// TwinCAT 3 PLC project PRG_HMIElements
// Title: B_HMIElements
// Company: RafalOS
// Author: Rafał Osajda
// ProjectVersion: 0.0.0.4
// ProgramVersion: 3.1.4024.0
// libraries:
//   B_Base, * (RafalOS)
//   B_Base_HMI_Connector, * (RafalOS)
//   Tc2_Standard, * (Beckhoff Automation GmbH)
//   Tc2_System, * (Beckhoff Automation GmbH)
//   Tc3_Module, * (Beckhoff Automation GmbH)
// project tree:
//   GVLs/ GVL_HMIEConstans.TcGVL (not stored)
//   / PlcTask.TcTTO
//   POUs Compilation/ PRG_Compilation.TcPOU
//   POUs/01A_Button/ FB_HMIEButton.TcPOU, ITF_HMIEButton.TcIO (not stored), ITF_HMIEButton_HMI_Connector.TcIO, ITF_HMIEButton_HMI_Init.TcIO (not stored)
//   POUs/01B_ButtonHMI/ FB_HMIEButton_HMI.TcPOU, ITF_HMIEButton_HMI.TcIO
//   POUs/02A_Menu/ FB_HMIEMenu.TcPOU, ITF_HMIEMenu_HMI_Connector.TcIO, ITF_HMIEMenu_HMI_Init.TcIO, ITF_HMIEMenu.TcIO
//   POUs/02B_MenuHMI/ FB_HMIEMenu_HMI.TcPOU, ITF_HMIEMenu_HMI.TcIO

CONFIGURATION PRG_HMIElements
    RESOURCE PLC ON TwinCAT3
        TASK PlcTask(INTERVAL := T#10ms, PRIORITY := 20);
        PROGRAM PRG_Compilation WITH PlcTask : PRG_Compilation;
    END_RESOURCE
END_CONFIGURATION

// ---- POUs/01A_Button/ITF_HMIEButton_HMI_Connector.TcIO
(*			
	RafalOS
	Rafał Osajda		12.11.2025		TC 4024.66
	Zbiór metod umożliwiające odczyt danych z hmi 
*)
INTERFACE ITF_HMIEButton_HMI_Connector EXTENDS ITF_BaseComponent_HMI_Connector

END_INTERFACE

// ---- POUs/01B_ButtonHMI/ITF_HMIEButton_HMI.TcIO
(*			
	RafalOS
	Rafał Osajda		12.11.2025		TC 4024.66
	interfejs potrzebny w HMI
*)
INTERFACE ITF_HMIEButton_HMI EXTENDS ITF_BaseComponent_HMI

END_INTERFACE

// ---- POUs/02A_Menu/ITF_HMIEMenu_HMI_Connector.TcIO
(*			
	RafalOS
	Rafał Osajda		12.11.2025		TC 4024.66
	Zbiór metod umożliwiające odczyt danych z hmi 
*)
INTERFACE ITF_HMIEMenu_HMI_Connector EXTENDS ITF_BaseControlElement_HMI_Connector

END_INTERFACE

// ---- POUs/02A_Menu/ITF_HMIEMenu_HMI_Init.TcIO
(*			
	RafalOS
	Rafał Osajda		12.11.2025		TC 4024.66
	interfejs do przekazywania przy tworzeniu elementów
*)
INTERFACE ITF_HMIEMenu_HMI_Init EXTENDS ITF_BaseControlElement, ITF_HMIEMenu_HMI_Connector

END_INTERFACE

// ---- POUs/02A_Menu/ITF_HMIEMenu.TcIO
INTERFACE ITF_HMIEMenu EXTENDS ITF_BaseControlElement

METHOD PUBLIC GetNumberOfActriveScreen : INT
VAR_INPUT
END_VAR
END_METHOD

METHOD IsActiveButton : BOOL
VAR_INPUT
	iButton		: INT;	//numer przycisku
	bIN			: BOOL;
END_VAR
END_METHOD

METHOD PUBLIC IsChangePage : BOOL
VAR_INPUT
END_VAR
END_METHOD

METHOD IsEnableButton : BOOL
VAR_INPUT
	iButton		: INT;	//numer przycisku
	bIN			: BOOL;
END_VAR
END_METHOD

METHOD IsVisibleButton : BOOL
VAR_INPUT
	iButton		: INT;	//numer przycisku
	bIN			: BOOL;
END_VAR
END_METHOD

METHOD PUBLIC ResetChangePage
VAR_INPUT
END_VAR
END_METHOD

METHOD SetActiveButton : BOOL
VAR_INPUT
	iButton		: INT;	//numer przycisku
	bIN			: BOOL;
END_VAR
END_METHOD

METHOD SetEnableButton : BOOL
VAR_INPUT
	iButton		: INT;	//numer przycisku
	bIN			: BOOL;
END_VAR
END_METHOD

METHOD SetVisibleButton : BOOL
VAR_INPUT
	iButton		: INT;	//numer przycisku
	bIN			: BOOL;
END_VAR
END_METHOD

(*			
	RafalOS
	Rafał Osajda		11.11.2025		TC 4024.66
	testuje czy jest coś naciśnięte w menu i przełącza
*)
METHOD PUBLIC Testing : BOOL
END_METHOD

END_INTERFACE

// ---- POUs/02B_MenuHMI/ITF_HMIEMenu_HMI.TcIO
(*			
	RafalOS
	Rafał Osajda		12.11.2025		TC 4024.66
	interfejs potrzebny w HMI
*)
INTERFACE ITF_HMIEMenu_HMI EXTENDS ITF_BaseComponent_HMI

END_INTERFACE

// ---- POUs Compilation/PRG_Compilation.TcPOU
PROGRAM PRG_Compilation
VAR
	fbButton		: FB_HMIEButton;
	fbButtonHMI		: FB_HMIEButton_HMI (itfButton := fbButton);
	fbMenu			: FB_HMIEMenu;
	fbMenuHMI		: FB_HMIEMenu_HMI (itfMenu := fbMenu);
END_VAR

END_PROGRAM

// ---- POUs/01A_Button/FB_HMIEButton.TcPOU
FUNCTION_BLOCK FB_HMIEButton EXTENDS FB_BaseComponent IMPLEMENTS ITF_HMIEButton, ITF_HMIEButton_HMI_Init
VAR
	bContact			: BOOL;
	bActive				: BOOL;	//wybrany
	bVisible			: BOOL; //widoczny
	bEnable				: BOOL; //wlaczony
END_VAR

METHOD PUBLIC IsActive : BOOL
VAR_INPUT
END_VAR
IsActive		:= THIS^.bActive;
END_METHOD

METHOD PUBLIC IsEnable : BOOL
VAR_INPUT
END_VAR
IsEnable		:= THIS^.bEnable;
END_METHOD

METHOD PUBLIC IsPressed : BOOL
VAR_INPUT
END_VAR
IsPressed		:= THIS^.bContact;
END_METHOD

METHOD PUBLIC IsVisible : BOOL
VAR_INPUT
END_VAR
IsVisible		:= THIS^.bVisible;
END_METHOD

METHOD PUBLIC SetActive
VAR_INPUT
	bIN: BOOL;
END_VAR
THIS^.bActive		:= bIN;
END_METHOD

METHOD PUBLIC SetEnable
VAR_INPUT
	bIN: BOOL;
END_VAR
THIS^.bEnable		:= bIN;
END_METHOD

METHOD PUBLIC SetPressed
VAR_INPUT
	bIN: BOOL;
END_VAR
THIS^.bContact		:= bIN;
END_METHOD

METHOD PUBLIC SetVisible
VAR_INPUT
	bIN: BOOL;
END_VAR
THIS^.bVisible		:= bIN;
END_METHOD

END_FUNCTION_BLOCK

// ---- POUs/01B_ButtonHMI/FB_HMIEButton_HMI.TcPOU
FUNCTION_BLOCK FB_HMIEButton_HMI EXTENDS FB_BaseComponent_HMI IMPLEMENTS ITF_HMIEButton_HMI
VAR
	itfButton			: ITF_HMIEButton_HMI_Connector;
END_VAR

METHOD FB_init : BOOL
VAR_INPUT
	bInitRetains : BOOL; // if TRUE, the retain variables are initialized (warm start / cold start)
	bInCopyCode : BOOL;  // if TRUE, the instance afterwards gets moved into the copy code (online change)
	itfButton			: ITF_HMIEButton_HMI_Init;
END_VAR
THIS^.itfButton := itfButton;
//Przypisanie do elementów z biblioteki
THIS^.itfBaseLoggerElementConnector		:= itfbutton;
THIS^.itfBaseComponentConnector			:= itfbutton;

//
THIS^.itfBaseLoggerConnector			:= itfBaseLoggerConnector;

IF (THIS^.itfButton <> 0 AND
	THIS^.itfBaseLoggerElementConnector <> 0 AND
	THIS^.itfBaseComponentConnector	<> 0 AND
	THIS^.itfBaseLoggerConnector <> 0) THEN
	THIS^.bIsInit						:= TRUE;
END_IF
END_METHOD

END_FUNCTION_BLOCK

// ---- POUs/02A_Menu/FB_HMIEMenu.TcPOU
FUNCTION_BLOCK FB_HMIEMenu EXTENDS FB_BaseControlElement IMPLEMENTS ITF_HMIEMenu, ITF_HMIEMenu_HMI_Init
VAR
	arrButtons				: ARRAY [0..GVL_HMIEConstans.MAX_NUMBER_OF_BUTTON_IN_MENU] OF ITF_HMIEButton;
	iNumberOfButton			: INT := -1;	//ilosć przycisków w menu
	iActiveButton			: INT;	//numer aktywnego przycisku
	iActiveButtonPrev		: INT;
	bChangePage				: BOOL; //zmiana strony
END_VAR

METHOD PUBLIC AddButton : BOOL
VAR_INPUT
	fbButton			: ITF_HMIEButton;
END_VAR
IF (THIS^.iNumberOfButton + 1 <= GVL_HMIEConstans.MAX_NUMBER_OF_BUTTON_IN_MENU) THEN
	THIS^.iNumberOfButton := THIS^.iNumberOfButton + 1;
	THIS^.arrButtons [THIS^.iNumberOfButton] := fbButton;
	THIS^.arrButtons [THIS^.iNumberOfButton].SetEnable (bIN := TRUE);
	THIS^.arrButtons [THIS^.iNumberOfButton].SetVisible (bIN := TRUE);
	THIS^.AddComponent (itfComponent := fbButton);
	AddButton := TRUE;
ELSE
	AddButton := FALSE;
END_IF
END_METHOD

METHOD PUBLIC GetNumberOfActrivePreviewScreen : INT
VAR_INPUT
END_VAR
GetNumberOfActrivePreviewScreen := THIS^.iActiveButtonPrev;
END_METHOD

METHOD PUBLIC GetNumberOfActriveScreen : INT
VAR_INPUT
END_VAR
GetNumberOfActriveScreen := THIS^.iActiveButton;
END_METHOD

METHOD PUBLIC GetTitleOfActivePage : WSTRING
VAR_INPUT
END_VAR
//GetTitleOfActivePage := this^.arrButtons [this^.iActiveButton].GetName ();
END_METHOD

METHOD IsActiveButton : BOOL
VAR_INPUT
	iButton		: INT;	//numer przycisku
	bIN			: BOOL;
END_VAR
IsActiveButton	:= THIS^.arrButtons [iButton].IsActive ();
END_METHOD

METHOD PUBLIC IsChangePage : BOOL
VAR_INPUT
END_VAR
IsChangePage := THIS^.bChangePage;
END_METHOD

METHOD IsEnableButton : BOOL
VAR_INPUT
	iButton		: INT;	//numer przycisku
	bIN			: BOOL;
END_VAR
IsEnableButton	:= THIS^.arrButtons [iButton].IsEnable ();
END_METHOD

METHOD IsVisibleButton : BOOL
VAR_INPUT
	iButton		: INT;	//numer przycisku
	bIN			: BOOL;
END_VAR
IsVisibleButton	:= THIS^.arrButtons [iButton].IsVisible ();
END_METHOD

METHOD PUBLIC ResetChangePage
VAR_INPUT
END_VAR
THIS^.bChangePage := FALSE;
END_METHOD

METHOD SetActiveButton : BOOL
VAR_INPUT
	iButton		: INT;	//numer przycisku
	bIN			: BOOL;
END_VAR
THIS^.arrButtons [iButton].SetActive (bIN := bIN);
END_METHOD

METHOD SetEnableButton : BOOL
VAR_INPUT
	iButton		: INT;	//numer przycisku
	bIN			: BOOL;
END_VAR
THIS^.arrButtons [iButton].SetEnable (bIN := bIN);
END_METHOD

METHOD SetVisibleButton : BOOL
VAR_INPUT
	iButton		: INT;	//numer przycisku
	bIN			: BOOL;
END_VAR
THIS^.arrButtons [iButton].SetVisible (bIN := bIN);
END_METHOD

(*			
	RafalOS
	Rafał Osajda		11.11.2025		TC 4024.66
	testuje czy jest coś naciśnięte w menu i przełącza
*)
METHOD PUBLIC Testing : BOOL
VAR
	iI		: INT;
	iJ		: INT;
END_VAR
FOR iI := 0 TO THIS^.iNumberOfButton DO
	IF (THIS^.arrButtons [iI].IsPressed ()) THEN
		FOR iJ := 0 TO THIS^.iNumberOfButton DO 
			THIS^.arrButtons [iJ].SetActive (bIN := FALSE);
		END_FOR
		THIS^.arrButtons [iI].SetActive (bIN := TRUE);
		THIS^.iActiveButtonPrev := THIS^.iActiveButton;
		THIS^.iActiveButton := iI;
		THIS^.bChangePage := TRUE;
	END_IF
END_FOR
END_METHOD

END_FUNCTION_BLOCK

// ---- POUs/02B_MenuHMI/FB_HMIEMenu_HMI.TcPOU
FUNCTION_BLOCK FB_HMIEMenu_HMI EXTENDS FB_BaseControlElement_HMI IMPLEMENTS ITF_HMIEMenu_HMI
VAR
	itfMenu			: ITF_HMIEMenu_HMI_Connector;
END_VAR

METHOD PUBLIC AddButton : BOOL
VAR_INPUT
	fbButtonHMI			: ITF_HMIEButton_HMI;
END_VAR
THIS^.AddComponent (itfComponentHMI := fbButtonHMI);
END_METHOD

METHOD FB_init : BOOL
VAR_INPUT
	bInitRetains : BOOL; // if TRUE, the retain variables are initialized (warm start / cold start)
	bInCopyCode : BOOL;  // if TRUE, the instance afterwards gets moved into the copy code (online change)
	itfMenu			: ITF_HMIEMenu_HMI_Init;
END_VAR
THIS^.itfMenu := itfMenu;

//Przypisanie do elementów z biblioteki
THIS^.itfBaseLoggerElementConnector		:= itfMenu;
THIS^.itfBaseComponentConnector			:= itfMenu;
THIS^.itfBaseControlElementConnector	:= itfMenu;
//
THIS^.itfBaseLoggerConnector			:= itfBaseLoggerConnector;
//

IF (THIS^.itfMenu <> 0 AND
	THIS^.itfBaseLoggerElementConnector <> 0 AND
	THIS^.itfBaseComponentConnector	<> 0 AND
	THIS^.itfBaseControlElementConnector <> 0 AND
	THIS^.itfBaseLoggerConnector <> 0) THEN
	THIS^.bIsInit						:= TRUE;
END_IF
END_METHOD

END_FUNCTION_BLOCK
